// TwinCAT 3 PLC project w4TrafficLight
// ProgramVersion: 3.1.4023.0
// libraries:
//   CmpBitmapPool, * (System)
//   Tc2_Standard, * (Beckhoff Automation GmbH)
//   Tc2_System, * (Beckhoff Automation GmbH)
//   Tc3_Module, * (Beckhoff Automation GmbH)
//   VisuSymbols,3.5.10.0,System
// project tree:
//   DUTs/ ST_TrafficLightInput.TcDUT, ST_TrafficLightOutput.TcDUT
//   / GlobalImagePool.TcGIPO (not stored), GlobalTextList.TcGTLO, PlcTask.TcTTO, Visualization Manager.TcVMO (not stored)
//   GVLs/ ImagePool.TcIPO (not stored), TrafficLightGVL.TcGVL, TrafficLightV1.TcVIS, TrafficLightVPrototype.TcVIS
//   POUs/ FB_Blinker.TcPOU, FB_Crossing.TcPOU, FB_TrafficLight.TcPOU, MAIN.TcPOU

CONFIGURATION w4TrafficLight
    RESOURCE PLC ON TwinCAT3
        TASK PlcTask(INTERVAL := T#10ms, PRIORITY := 20);
        PROGRAM MAIN WITH PlcTask : MAIN;
    END_RESOURCE
END_CONFIGURATION

// ---- DUTs/ST_TrafficLightInput.TcDUT
TYPE ST_TrafficLightInput :
STRUCT

	bDayMode : BOOL;
	bSetRed : BOOL;
	bSetGreen : BOOL;
END_STRUCT
END_TYPE

// ---- DUTs/ST_TrafficLightOutput.TcDUT
TYPE ST_TrafficLightOutput :
STRUCT
	bRed : BOOL;
	bYellow : BOOL;
	bGreen : BOOL;
	
END_STRUCT
END_TYPE

// ---- GVLs/TrafficLightGVL.TcGVL
{attribute 'qualified_only'}
VAR_GLOBAL

	stTrafficInArray : ARRAY[1..4] OF ST_TrafficLightInput;
	stTrafficOutArray : ARRAY[1..4] OF ST_TrafficLightOutput;

END_VAR

// ---- POUs/MAIN.TcPOU
PROGRAM MAIN
VAR
	
	fbCrossing1 : FB_Crossing;
	(*
	bBool AT%I* : BOOL;
	bBool2 AT%Q* : BOOL;
	nInt1 AT%I* : INT;
	nInt12 AT%Q* : INT;
	nInt13 AT%Q* : INT;
	rTrig : R_TRIG;
	
*)
	
	

END_VAR



fbCrossing1();
(*
rTrig(CLK := bBool);
IF rTrig.Q THEN
	bBool2 := NOT bBool2;
END_IF
*)

END_PROGRAM

// ---- POUs/FB_Crossing.TcPOU
FUNCTION_BLOCK FB_Crossing
VAR_INPUT
	bCDayMode : BOOL;
	stMainIn : ST_TrafficLightInput;
	stSubIn : ST_TrafficLightInput;
END_VAR
VAR_OUTPUT
END_VAR
VAR
	fbTrafficLightArray : ARRAY[1..4] OF FB_TrafficLight; //defining the array
	idx : INT;
	tonCrossing : TON;
	nStep : INT;
	
END_VAR


CASE nStep OF
	
	0:  IF NOT bCDayMode THEN
			stMainIn.bDayMode := FALSE;
			stSubIn.bDayMode := FALSE;
		ELSE 
			stMainIn.bDayMode := TRUE;
			stSubIn.bDayMode := TRUE;
			nStep := 10;
		END_IF
	10: stMainIn.bSetRed := TRUE;
		stSubIn.bSetRed := TRUE;
		tonCrossing(IN := TRUE, PT := T#3S);
		IF tonCrossing.Q AND bCDayMode THEN
			stMainIn.bSetRed := FALSE;
			stSubIn.bSetRed := FALSE;
			tonCrossing(IN := FALSE);
			nStep := 20;
		END_IF
		IF NOT bCDayMode THEN
			tonCrossing(IN := FALSE);
			stMainIn.bSetGreen := TRUE;
			stMainIn.bSetRed := FALSE;
			stSubIn.bSetGreen := TRUE;
			stSubIn.bSetRed := FALSE;
			nStep := 0;
		END_IF
	20: stSubIn.bSetRed := TRUE;
		IF fbTrafficLightArray[3].stTrafficLightOutput.bRed THEN
			stMainIn.bSetGreen := TRUE;
		END_IF
		tonCrossing(IN := TRUE, PT := T#10S);
		IF tonCrossing.Q AND bCDayMode THEN
			tonCrossing(IN := FALSE);
			stMainIn.bSetGreen := FALSE;
			stSubIn.bSetRed := FALSE;
			nStep := 30;
		END_IF
		IF NOT bCDayMode THEN
			tonCrossing(IN := FALSE);
			stMainIn.bSetGreen := FALSE;
			stSubIn.bSetGreen := FALSE;
			nStep := 0;
		END_IF
	30: stMainIn.bSetRed := TRUE;
		IF fbTrafficLightArray[1].stTrafficLightOutput.bRed THEN
			stSubIn.bSetGreen := TRUE;
		END_IF
		tonCrossing(IN := TRUE, PT := T#10S);
		IF tonCrossing.Q AND bCDayMode THEN
			tonCrossing(IN := FALSE);
			stMainIn.bSetRed := FALSE;
			stSubIn.bSetGreen := FALSE;
			nStep := 20;
		END_IF
		IF NOT bCDayMode THEN
			tonCrossing(IN := FALSE);
			stMainIn.bSetGreen := FALSE;
			stSubIn.bSetGreen := FALSE;
			nStep := 0;
		END_IF
			
	
END_CASE

FOR idx := 1 TO 2 DO    
			fbTrafficLightArray[idx](stTrafficLightInput := stMainIn);
END_FOR
FOR idx := 3 TO 4 DO    
			fbTrafficLightArray[idx](stTrafficLightInput := stSubIn);
END_FOR

END_FUNCTION_BLOCK

// ---- POUs/FB_TrafficLight.TcPOU
FUNCTION_BLOCK FB_TrafficLight
VAR_INPUT
	//bDayMode : BOOL;
	//bSetRed : BOOL;
	//bSetGreen : BOOL;
	stTrafficLightInput : ST_TrafficLightInput;
END_VAR
VAR_OUTPUT
	//bRed : BOOL;
	//bYellow : BOOL;
	//bGreen : BOOL;
	stTrafficLightOutput : ST_TrafficLightOutput;
END_VAR
VAR
	nStep : INT := 0;
	fbBlinker : FB_Blinker;
	//tonRedTimer : TON;
	tonYellowTimer : TON;
	//tonGreenTimer : TON;
	rTrigSetGreen : R_TRIG;
	rTrigSetRed : R_TRIG;
END_VAR

CASE nStep OF
	0: 	IF NOT stTrafficLightInput.bDayMode THEN
			fbBlinker(bEnable := TRUE, bBlink => stTrafficLightOutput.bYellow);
		ELSE
			fbBlinker(bEnable := FALSE);
			stTrafficLightOutput.bYellow := FALSE;
			nStep := 10;
		END_IF
	10: stTrafficLightOutput.bRed := TRUE;
		stTrafficLightOutput.bYellow := FALSE;
		stTrafficLightOutput.bGreen := FALSE;
		//tonRedTimer(IN:= TRUE, PT := T#10S);
		IF NOT stTrafficLightInput.bDayMode THEN
			stTrafficLightOutput.bRed := FALSE;
			stTrafficLightOutput.bGreen := FALSE;
			nStep := 0;
		END_IF
		rTrigSetGreen(CLK := stTrafficLightInput.bSetGreen);
		IF rTrigSetGreen.Q THEN
			//tonRedTimer(IN := FALSE);//reset my timer
			nStep := 20;
		END_IF
	20: stTrafficLightOutput.bRed := TRUE;
		stTrafficLightOutput.bYellow := TRUE;
		stTrafficLightOutput.bGreen := FALSE;
		tonYellowTimer(in:= TRUE, PT := T#3S);		
		IF tonYellowTimer.Q THEN
			tonYellowTimer(IN := FALSE);
			nStep := 30;
		END_IF
		IF NOT stTrafficLightInput.bDayMode THEN
			tonYellowTimer(IN := FALSE);
			stTrafficLightOutput.bRed := FALSE;
			stTrafficLightOutput.bGreen := FALSE;
			nStep := 0;
		END_IF
	30: stTrafficLightOutput.bRed := FALSE;
		stTrafficLightOutput.bYellow := FALSE;
		stTrafficLightOutput.bGreen := TRUE;
		//tonGreenTimer(IN := TRUE, PT := T#10S);
		rTrigSetRed(CLK := stTrafficLightInput.bSetRed);
		IF rTrigSetRed.Q THEN
			//tonGreenTimer(IN := FALSE);
			nStep := 40;
		END_IF
		IF NOT stTrafficLightInput.bDayMode THEN
			stTrafficLightOutput.bRed := FALSE;
			stTrafficLightOutput.bGreen := FALSE;
			nStep := 0;
		END_IF
	40: stTrafficLightOutput.bRed := FALSE;
		stTrafficLightOutput.bYellow := TRUE;
		stTrafficLightOutput.bGreen := FALSE;
		tonYellowTimer(in:= TRUE, PT := T#3S);
		IF tonYellowTimer.Q THEN
			tonYellowTimer(IN := FALSE);
			nStep := 10;
		END_IF
		IF NOT stTrafficLightInput.bDayMode THEN
			tonYellowTimer(IN := FALSE);
			nStep := 0;
		END_IF
END_CASE

END_FUNCTION_BLOCK

// ---- POUs/FB_Blinker.TcPOU
FUNCTION_BLOCK FB_Blinker
VAR_INPUT
	bEnable : BOOL;
END_VAR
VAR_OUTPUT
	bBlink : BOOL;
END_VAR
VAR
	tonTimer1 : TON;
	tonTimer2 : TON;
END_VAR

IF bEnable AND NOT tonTimer2.Q THEN
	tonTimer1.IN := TRUE;
ELSE 
	tonTimer1.IN := FALSE;
END_IF

tonTimer1(PT := T#1000MS);

IF tonTimer1.Q THEN
	tonTimer2.IN := TRUE;
ELSE
	tonTimer2.IN := FALSE;
END_IF

tonTimer2(PT := T#1000MS);
bBlink := tonTimer1.Q;

END_FUNCTION_BLOCK

// ---- GlobalTextList.TcGTLO
TEXTLIST GlobalTextList
  59 = 'set Day Mode'
  780 = 'set Green'
  459 = 'Set Red'
  426 = 'set the day night mode'
END_TEXTLIST

// ---- GVLs/TrafficLightV1.TcVIS
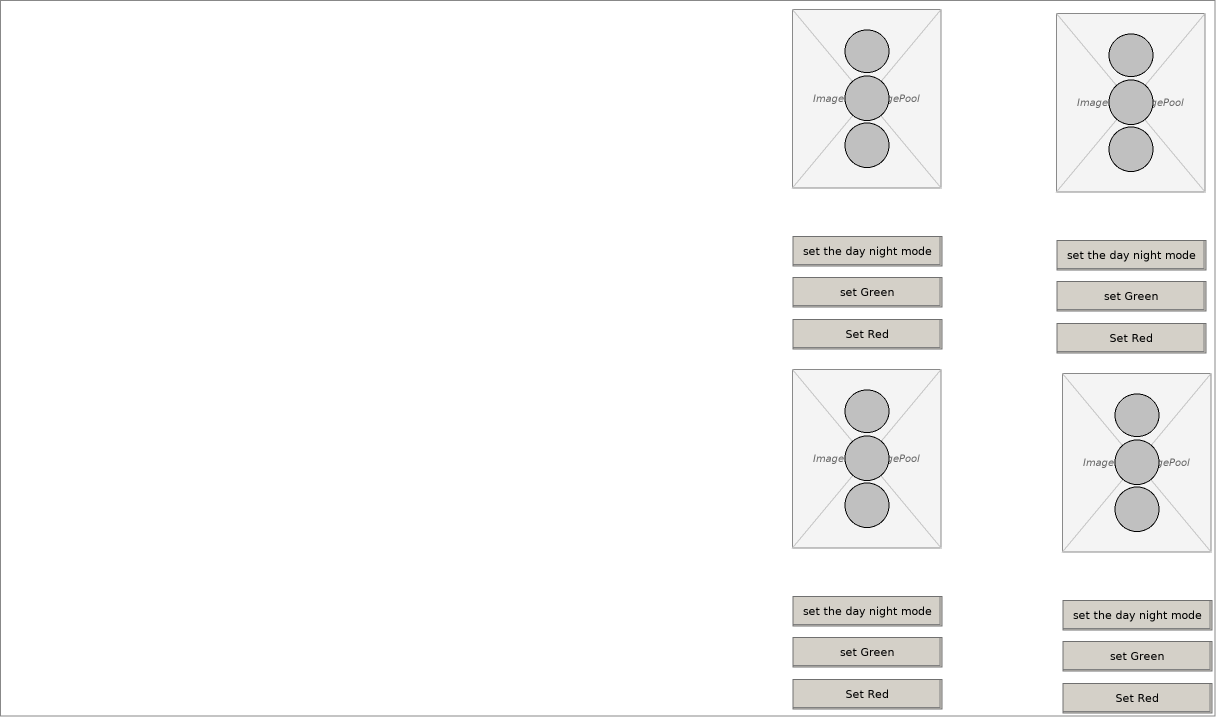
VISUALIZATION TrafficLightV1  // 1216x717
    Frame (792,369 152x342)
        shows TrafficLightVPrototype(stTrafficOut := MAIN.fbCrossing1.fbTrafficLightArray[1].stTrafficLightOutput)
    Frame (1062,373 152x342)
        shows TrafficLightVPrototype(stTrafficOut := MAIN.fbCrossing1.fbTrafficLightArray[3].stTrafficLightOutput)
    Frame (792,9 152x342)
        shows TrafficLightVPrototype(stTrafficOut := MAIN.fbCrossing1.fbTrafficLightArray[4].stTrafficLightOutput)
    Frame (1056,13 152x342)
        shows TrafficLightVPrototype(stTrafficOut := MAIN.fbCrossing1.fbTrafficLightArray[2].stTrafficLightOutput)
END_VISUALIZATION

// ---- GVLs/TrafficLightVPrototype.TcVIS
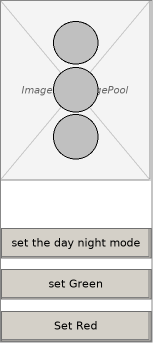
VISUALIZATION TrafficLightVPrototype  // 153x343
VAR_IN_OUT
	stTrafficIn : ST_TrafficLightInput;
	stTrafficOut : ST_TrafficLightOutput;
END_VAR
    Image (0,0 150x180), image: ImagePool.ImagePool
    Ellipse (53,67 45x45), colour toggle: stTrafficOut.bYellow
    Ellipse (53,21 45x43), colour toggle: stTrafficOut.bRed
    Ellipse (53,114 45x45), colour toggle: stTrafficOut.bGreen
    Button (1,228 150x30), "set the day night mode"
        toggle MAIN.fbCrossing1.bCDayMode
    Button (1,269 150x30), "set Green"
        tap stTrafficIn.bSetGreen
    Button (1,311 150x30), "Set Red"
        tap stTrafficIn.bSetRed
END_VISUALIZATION
